// TIA Portal V19 export
FUNCTION "Cont_PQI" : Void   // FC150, STL
TITLE = control PQI-byte
{ S7_Optimized_Access := 'TRUE' }
AUTHOR : fur
FAMILY : FC
NAME : FC50
// stored: AutoNumber false
   VAR_INPUT
      IB_PQI : Byte;   // Input PQI-byte
   END_VAR
   VAR_OUTPUT
      O_DI4 : Bool;   // Output signal status Pin 4
      O_DI2 : Bool;   // Output signal status Pin 2
      O_DA : Bool;   // Output device recognized
      O_DE : Bool;   // Output device error event has appeared
      O_PQ : Bool;   // Output port qualifer process data valid
   END_VAR
   VAR_TEMP
      TW_Flag : Word;
   END_VAR
BEGIN

NETWORK
TITLE = 
      L     #IB_PQI;
      T     #TW_Flag;

      L     #TW_Flag;
      L     1;
      AW;
      L     1;
      ==I;
      =     #O_DI4;



      L     #TW_Flag;
      L     2;
      AW;
      L     2;
      ==I;
      =     #O_DI2;

      L     #TW_Flag;
      L     32;
      AW;
      L     32;
      ==I;
      =     #O_DA;

      L     #TW_Flag;
      L     64;
      AW;
      L     64;
      ==I;
      =     #O_DE;


      L     #TW_Flag;
      L     128;
      AW;
      L     128;
      ==I;
      =     #O_PQ;

END_FUNCTION
